// TIA Portal V18 export
// export: Created 2026-06-12T02:00:00Z, ExportSetting WithDefaults
VAR_GLOBAL   // PLC tag table "PLC_AI_B7_Tags"
   AI_B7_K03_PT02_Pressure AT %MD800 : Real;   // PRESSURE 7-8 bar
   AI_B7_K03_TT04_Temp AT %MD804 : Real;   // TEMP 50-80 °C
   AI_B7_K03_TT05_Temp AT %MD808 : Real;   // TEMP 50-80 °C
   AI_B7_K03_TT06_Temp AT %MD812 : Real;   // TEMP 50-80 °C
   AI_B7_K03_TT07_Temp AT %MD816 : Real;   // TEMP 50-80 °C
   AI_B7_K03_PT07_Pressure AT %MD820 : Real;   // PRESSURE 7-8 bar
   AI_B7_K03_FT03_Flow AT %MD824 : Real;   // FLOW 100-200 L/h
   AI_B7_K03_Density_1 AT %MD828 : Real;   // COUNT 800-1000 kg/m3
   AI_B7_K03_LT01_Level AT %MD832 : Real;   // LEVEL 20-80 cm
   AI_B7_K03_LT02_Level AT %MD836 : Real;   // LEVEL 20-80 cm
   AI_B7_K03_TT01_Temp AT %MD840 : Real;   // TEMP 50-80 °C
   AI_B7_K03_TT02_Temp AT %MD844 : Real;   // TEMP 50-80 °C
   AI_B7_Reboiler_PV AT %MD848 : Real;   // FLOW 100-200 L/h
   AI_B7_Reboiler_SP AT %MD852 : Real;   // FLOW 100-200 L/h
   AI_B7_Reboiler_CV AT %MD856 : Real;   // PERCENT 20-80 %
   AI_B7_HE03_Primary_Temp AT %MD860 : Real;   // TEMP 50-80 °C
   AI_B7_HE03_Secondary_Temp AT %MD864 : Real;   // TEMP 50-80 °C
   AI_B7_K03_L08_Level AT %MD868 : Real;   // LEVEL 20-80 cm
   AI_B7_K03_L06_Level AT %MD872 : Real;   // LEVEL 20-80 cm
   AI_B7_K03_L05_Level AT %MD876 : Real;   // LEVEL 20-80 cm
   AI_B7_K03_L07_Level AT %MD880 : Real;   // LEVEL 20-80 cm
   AI_B7_K03_L04_Level AT %MD884 : Real;   // LEVEL 20-80 cm
   AI_B7_K03_L03_Level AT %MD888 : Real;   // LEVEL 20-80 cm
   AI_B7_V03A_Density AT %MD892 : Real;   // COUNT 800-1000 kg/m3
   AI_B7_Kettle_Flow_SP AT %MD896 : Real;   // FLOW 100-200 kg/h
   AI_B7_Keboiler_Flow_SP AT %MD900 : Real;   // FLOW 100-200 kg/h
   AI_B7_Reflux_Time_SP AT %MD904 : Real;   // COUNT 0-60 Min
   AI_B7_Time_Remain AT %MD908 : Real;   // COUNT 0-60 Min
   AI_B7_RD_Level_SP AT %MD912 : Real;   // LEVEL 20-80 cm
   AI_B7_Reflux_Flow_SP AT %MD916 : Real;   // FLOW 100-200 L/h
   AI_B7_Collection_SP AT %MD920 : Real;   // FLOW 100-200 L/h
   AI_B7_Total_Flowrate AT %MD924 : Real;   // FLOW 100-200 L/h
   AI_B7_ML_Qty_SP AT %MD928 : Real;   // COUNT 0-600 L
   AI_B7_ML_Qty_Total AT %MD932 : Real;   // COUNT 0-600 L
   AI_B7_Material_Code AT %MD936 : Real;   // COUNT 0-99
   AI_B7_Stage_Number AT %MD940 : Real;   // COUNT 0-20
   AI_B7_Batch_Number AT %MD944 : Real;   // COUNT 0-9999
   AI_B7_Current_User_ID AT %MD948 : Real;   // COUNT 0-999
   AI_B7_K_05_L_704_HI AT %MD952 : Real;   // LEVEL 20-80 cm
   AI_B7_Density_SP AT %MD956 : Real;   // COUNT 800-1000 kg/m3
   AI_B7_CTS_Flow_1 AT %MD960 : Real;   // FLOW 100-200 kg/h
   AI_B7_CTS_Flow_2 AT %MD964 : Real;   // FLOW 100-200 kg/h
   AI_B7_Steam_PT01_Temp AT %MD968 : Real;   // TEMP 50-80 °C
   AI_B7_Steam_PT02_Temp AT %MD972 : Real;   // TEMP 50-80 °C
   AI_B7_CWS_TT01_Temp AT %MD976 : Real;   // TEMP 50-80 °C
   AI_B7_CWS_TT02_Temp AT %MD980 : Real;   // TEMP 50-80 °C
   AI_B7_CWS_TT03_Temp AT %MD984 : Real;   // TEMP 50-80 °C
   AI_B7_CWAR_TT01_Temp AT %MD988 : Real;   // TEMP 50-80 °C
   AI_B7_CWAR_TT02_Temp AT %MD992 : Real;   // TEMP 50-80 °C
   AI_B7_CWAR_TT03_Temp AT %MD996 : Real;   // TEMP 50-80 °C
   AI_B7_CWAR_TT04_Temp AT %MD1000 : Real;   // TEMP 50-80 °C
   AI_B7_K03_CV01_PV AT %MD1004 : Real;   // PERCENT 20-80 %
   AI_B7_K03_CV01_SP AT %MD1008 : Real;   // PERCENT 20-80 %
   AI_B7_K03_CV01_CV AT %MD1012 : Real;   // PERCENT 20-80 %
   AI_B7_Steam_CV01_PV AT %MD1016 : Real;   // PERCENT 20-80 %
   AI_B7_Steam_CV01_SP AT %MD1020 : Real;   // PERCENT 20-80 %
   AI_B7_Steam_CV01_CV AT %MD1024 : Real;   // PERCENT 20-80 %
   AI_B7_K03_Jacket_PV AT %MD1028 : Real;   // TEMP 50-80 °C
   AI_B7_K03_Jacket_SP AT %MD1032 : Real;   // TEMP 50-80 °C
   AI_B7_K03_Jacket_CV AT %MD1036 : Real;   // PERCENT 20-80 %
   AI_B7_CHWR_TT01_Temp AT %MD1040 : Real;   // TEMP 50-80 °C
   AI_B7_CHWR_TT02_Temp AT %MD1044 : Real;   // TEMP 50-80 °C
   AI_B7_CHWS_TT01_Temp AT %MD1048 : Real;   // TEMP 50-80 °C
   AI_B7_CHWS_TT02_Temp AT %MD1052 : Real;   // TEMP 50-80 °C
   AI_B7_K03_TT03_Temp AT %MD1056 : Real;   // TEMP 50-80 °C
END_VAR
